{attribute 'qualified_only' := ''}
{attribute 'strict' := ''}
TYPE eAdasKom_State :
(
	WaitForNC,
	SetDefaultkonfig,
	Running,
	Error
);
END_TYPE

(* stored: Version 1.1.0.1, ProductVersion 3.1.4022.16
   DUT eAdasKom_State: Id {f573dd93-929e-486d-8d34-7148881e6277} *)
